INTERFACE ITF_Vacuumzuignap

METHOD Loslaten : BOOL
VAR_INPUT
END_VAR
END_METHOD

METHOD Oppakken : BOOL
VAR_INPUT
END_VAR
END_METHOD

PROPERTY Status : E_VacuumzuignapStatus
GET
END_GET
SET
END_SET
END_PROPERTY

END_INTERFACE

(* stored: Version 1.1.0.1
   Itf ITF_Vacuumzuignap: Id {0df57663-b1aa-49e9-991c-c46e280631c2}
   Method Loslaten: Id {84f6da63-5f77-42c2-8fe3-8a35ca9637b2}
   Method Oppakken: Id {1c743885-6b76-4c87-9e20-2708cc9ed8a9}
   Property Status: Id {24e3e0b3-092b-4d54-a409-6722d1e34c45}
   Get Get: Id {d28ad8a0-d2a1-4b03-9966-9716d44f9284}
   Set Set: Id {b04cb878-523f-4452-b240-038ec4c5a8b9} *)
